// TwinCAT 3 PLC project Project1
// ProgramVersion: 3.1.4022.3
// libraries:
//   Tc2_Standard, * (Beckhoff Automation GmbH)
//   Tc2_System, * (Beckhoff Automation GmbH)
//   Tc3_Module, * (Beckhoff Automation GmbH)
// project tree:
//   GVLs/ GVL.TcGVL
//   / PlcTask.TcTTO
//   POUs/ AdditionFunction.TcPOU, DoSomeMath.TcPOU, Fakultaet.TcPOU, MAIN.TcPOU, SubtractionFunction.TcPOU
// real-time tasks:
//   TASK PlcTask: cycle T#5ms, priority 20, ADS port 350
// I/O:
//   DEVICE Gerät 1 (EtherCAT), AmsNetId 5.12.140.184.2.1
//     Klemme 1 (EK1200) [EK1200-5000 EtherCAT Netzteil (2A E-Bus)]
//       Klemme 2 (EL1004) [EL1004 4K. Dig. Eingang 24V, 3ms]
//       Klemme 3 (EL2004) [EL2004 4K. Dig. Ausgang 24V, 0.5A]
//       Klemme 4 (EL3004) [EL3004 4K.Ana. Eingang  +/-10V]
//       Klemme 5 (EL4034) [EL4034 4K. Ana. Ausgang +/-10V, 12bit]
//       Klemme 6 (EK1110) [EK1110 EtherCAT-Verlängerung]
// variable links:
//   Project1/Project1 Instance <-> Device 1 (EtherCAT)/Term 1 (EK1200)/Term 2 (EL1004)
//     PlcTask Inputs/GVL.globButtonBlue <-> Channel 2/Input BlueButton
//     PlcTask Inputs/GVL.globButtonYellow <-> Channel 1/Input YellowButton
//   Project1/Project1 Instance <-> Device 1 (EtherCAT)/Term 1 (EK1200)/Term 3 (EL2004)
//     PlcTask Outputs/GVL.globLightGreen <-> Channel 2/OutputGreenLight
//     PlcTask Outputs/GVL.globLightRed <-> Channel 1/Output RedLight

CONFIGURATION Project1
    RESOURCE PLC ON TwinCAT3
        TASK PlcTask(INTERVAL := T#5ms, PRIORITY := 20);
        PROGRAM MAIN WITH PlcTask : MAIN;
    END_RESOURCE
END_CONFIGURATION

// ---- GVLs/GVL.TcGVL
{attribute 'qualified_only'}
VAR_GLOBAL
	globButtonYellow AT %I*: BOOL;
	globButtonBlue AT %I*: BOOL;
	globLightGreen AT %Q*: BOOL;
	globLightRed AT %Q*: BOOL;
END_VAR

// ---- POUs/MAIN.TcPOU
PROGRAM MAIN
VAR
	B_myByte : BYTE := 128;					// BYTE = 8 Bit Speicherplatz (0 bis 255)
	r_myReal : REAL := 0.0;			// INT = 16 Bit Speihcerplatz (-32768 bis 32767)
	ui_myUnsignedInteger : UINT := 5000;	// UINT = 16 Bit Speicherplatz (0 bis 65535)	
	w_myWord : WORD := 65535;				// WORD = 16 Bit Speicherplatz (0 bis 65535)
	b_myBool : BOOL := TRUE;				// BOOL = 8 Bit Speicherplatz
	i_valueA: REAL;
	i_valueB: REAL;
	i_myResultMinus: INT;
	l_resultFak: LINT;
	i_counterYellow : INT := 0;
	i_counterBlue : INT := 0;
END_VAR

B_myByte := 100;

//r_myReal := AdditionFunction(i_valueA := 12.43, i_valueB := 1.02);
//i_myResultMinus := SubtractionFunction(i_valueA := 200, i_valueB := 20);
DoSomeMath(r_InputA := i_valueA := 12, r_InputB := 3.4);
l_resultFak := Fakultaet(i_fakultat := 10);

IF(GVL.globButtonYellow)
	THEN
	GVL.globLightGreen := TRUE;
	i_counterYellow := i_counterYellow +1;
	CASE i_counterYellow OF
		200 : ;
		400 : ;
		600 : ;
		800 :
		1000:
		1200:
		1400:
		1600:
		1800:
		2000:
END_CASE;
ELSE
	GVL.globLightGreen := FALSE;
END_IF

IF(GVL.globButtonBlue)
	THEN
	GVL.globLightRed := TRUE;
	i_counterBlue := i_counterBlue + 1;
ELSE
	GVL.globLightRed := FALSE;
END_IF

END_PROGRAM

// ---- POUs/DoSomeMath.TcPOU
PROGRAM DoSomeMath
VAR_INPUT
	r_InputA : REAL ;
	r_InputB : REAL ;
END_VAR
VAR
	r_ResultAdd : REAL;
	r_ResultSub : REAL;
END_VAR

r_ResultAdd := AdditionFunction(r_InputA, r_InputB);
r_ResultSub := SubtractionFunction(r_InputA, r_InputB);

END_PROGRAM

// ---- POUs/AdditionFunction.TcPOU
FUNCTION AdditionFunction : REAL
VAR_INPUT
	i_valueA : REAL;
	i_valueB : REAL;
END_VAR

AdditionFunction := i_valueA + i_valueB;

END_FUNCTION

// ---- POUs/SubtractionFunction.TcPOU
FUNCTION SubtractionFunction : REAL
VAR_INPUT
	i_valueA : REAL;
	i_valueB : REAL;
END_VAR
VAR
END_VAR

SubtractionFunction := i_valueA - i_valueB;

END_FUNCTION

// ---- POUs/Fakultaet.TcPOU
FUNCTION Fakultaet : LINT
VAR_INPUT
	i_fakultat : INT;
END_VAR
VAR
	l_result : LINT := 1;
	i : INT;
END_VAR

FOR i := 1 TO i_fakultat BY 1 DO
	IF(i_fakultat = 0)
		THEN
		l_result := 1;
		RETURN;
	END_IF
l_result := l_result * i;
END_FOR;
Fakultaet := l_result;

END_FUNCTION
